PROGRAM P_Task2
VAR
END_VAR

END_PROGRAM

(* stored: Version 1.1.0.1, ProductVersion 3.1.4024.12
   POU P_Task2: Id {9ed0eceb-1ce7-484d-b635-a4528063a015}, SpecialFunc None *)
